// TwinCAT 3 PLC project ArrayObjDemo
// ProgramVersion: 3.1.4023.0
// libraries:
//   Tc2_Standard, * (Beckhoff Automation GmbH)
//   Tc2_System, * (Beckhoff Automation GmbH)
//   Tc3_Module, * (Beckhoff Automation GmbH)
// project tree:
//   DUTs/ MotorInputVariables.TcDUT, MotorOutputVariables.TcDUT
//   / PlcTask.TcTTO
//   POUs/ MAIN.TcPOU, Motor.TcPOU, Plc_Prog.TcPOU
// real-time tasks:
//   TASK PlcTask: cycle T#10ms, priority 20, ADS port 350

CONFIGURATION ArrayObjDemo
    RESOURCE PLC ON TwinCAT3
        TASK PlcTask(INTERVAL := T#10ms, PRIORITY := 20);
        PROGRAM MAIN WITH PlcTask : MAIN;
    END_RESOURCE
END_CONFIGURATION

// ---- DUTs/MotorInputVariables.TcDUT
TYPE MotorInputVariables :
STRUCT
	Start : BOOL;
	Stop : BOOL;
	Oveload : BOOL;
END_STRUCT
END_TYPE

// ---- DUTs/MotorOutputVariables.TcDUT
TYPE MotorOutputVariables  :
STRUCT
	Coil : BOOL;
END_STRUCT
END_TYPE

// ---- POUs/MAIN.TcPOU
PROGRAM MAIN
VAR
END_VAR

Plc_Prog();

END_PROGRAM

// ---- POUs/Plc_Prog.TcPOU
PROGRAM Plc_Prog
VAR
	Motors : ARRAY[1..3] OF Motor;
	MotorsIn : ARRAY[1..3] OF MotorInputVariables;
	MotorsOut : ARRAY[1..3] OF MotorOutputVariables;
	
END_VAR

Motors[1](MotorInputs:=MotorsIn[1], MotorOutputs=>MotorsOut[1]);
Motors[2](MotorInputs:=MotorsIn[2], MotorOutputs=>MotorsOut[2]);
Motors[3](MotorInputs:=MotorsIn[3], MotorOutputs=>MotorsOut[3]);

END_PROGRAM

// ---- POUs/Motor.TcPOU
FUNCTION_BLOCK Motor
VAR_INPUT
	MotorInputs : MotorInputvariables;
END_VAR
VAR_OUTPUT
	MotorOutputs : MotorOutputVariables;
END_VAR
VAR
	Start : BOOL;
	Stop : BOOL;
END_VAR

Start := MotorInputs.Start;
Stop := MotorInputs.Stop;

IF Start AND Stop = FALSE AND MotorInputs.Oveload = FALSE THEN
	MotorOutputs.Coil := TRUE;
ELSE
	MotorOutputs.Coil := FALSE;
	
END_IF

END_FUNCTION_BLOCK
